FUNCTION_BLOCK FB_Motor_Test EXTENDS FB_TestSuite
VAR
    fbMotor : FB_MotorController;
END_VAR

StartWithNoFault_Test();
StartWithFault_Test();
Stop_Test();
FaultDuringRun_Test();
StopAfterFault_Test();

METHOD FaultDuringRun_Test
VAR_INPUT
END_VAR
 fbMotor.Stop(); 
fbMotor.Start(bFault := FALSE);  
fbMotor.Execute(bFault := TRUE);

Test('FaultDuringRun_Test');
   AssertFalse(
      Condition :=  fbMotor.IsRunning,
        Message   :=   'Motor should not run when there is fault');
			
TEST_FINISHED();
END_METHOD

METHOD StartWithFault_Test
VAR_INPUT
END_VAR

Test('StartWithFault_Test');
 fbMotor.Stop();
fbMotor.Start(bFault := TRUE);

   AssertFalse(
         Condition :=fbMotor.IsRunning,
         Message   :=  'Motor should not run when there is fault');
		
 fbMotor.Stop(); 
fbMotor.Start(bFault := FALSE);

   AssertTrue(
        Condition := fbMotor.IsRunning,
       Message   :=  'Motor should run when no fault');
				 
		 
TEST_FINISHED();
END_METHOD

METHOD StartWithNoFault_Test 
VAR_INPUT
	
END_VAR
 fbMotor.Stop(); 
fbMotor.Start(bFault := FALSE);

Test('StartWithNoFault_Test');
   AssertTrue(
        Condition := fbMotor.IsRunning,
       Message   :=  'Motor should run when no fault');
		
	
    TEST_FINISHED();
END_METHOD

METHOD Stop_Test
VAR_INPUT
END_VAR

 fbMotor.Start(bFault := FALSE);  
fbMotor.Stop();

Test('Stop_Test');
   AssertFalse(
        Condition := fbMotor.IsRunning,
         Message   :='Motor should not run when stopped is pressed');
		
TEST_FINISHED();
END_METHOD

METHOD StopAfterFault_Test 
VAR_INPUT
END_VAR
fbMotor.Stop();
    fbMotor.Execute(bFault := TRUE);    

  
    fbMotor.Start(bFault := TRUE);      // Try to restart with fault still on

    // ── Assert ────────────────────────────────────────────────
    TEST('StartWithActiveFault_MustStayStoped');
    AssertFalse(
        Condition := fbMotor.IsRunning,
        Message   := 'Motor must not restart while fault still active');
  
TEST_FINISHED();
END_METHOD

END_FUNCTION_BLOCK

(* stored: Version 1.1.0.1, ProductVersion 3.1.4024.16
   POU FB_Motor_Test: Id {3a16bd69-4871-43c6-a52d-075d93c717d7}, SpecialFunc None
   Method FaultDuringRun_Test: Id {ff1ee177-47dc-4396-9d9c-3faf7f54d771}
   Method StartWithFault_Test: Id {66b6cc70-e26c-44cd-bba3-5e78ea0e21b5}
   Method StartWithNoFault_Test: Id {f556bbaf-45e1-4112-8709-3e9032a57308}
   Method Stop_Test: Id {8ef5d4d5-9666-40fb-800f-c408e1821954}
   Method StopAfterFault_Test: Id {d393f69e-c48c-4acd-a8a7-c748c2ae80cd} *)
